(* Logix 5000 project; controller Ex_2_12 Emulate 5570 rev 33.11; software revision 33.00 *)
// Pallet lift table

TASK MainTask (continuous, watchdog 500 ms) : MainProgram

MODULES
   Local : Emulate 5570 (ICP 4, rev 33.11)
END_MODULES

VAR_GLOBAL   (* controller tags *)
   B1 : BOOL;   // Downward Sensor
   B2 : BOOL;   // Upward Sensor
   M1_Downward : BOOL;   // Actuator M1
   M1_Upward : BOOL;   // Actuator M1
   S1 : BOOL;   // Switch S1
   S2 : BOOL;   // Switch S2
END_VAR

PROGRAM MainProgram   (* main routine MainRoutine *)

ROUTINE MainRoutine   (* ladder *)
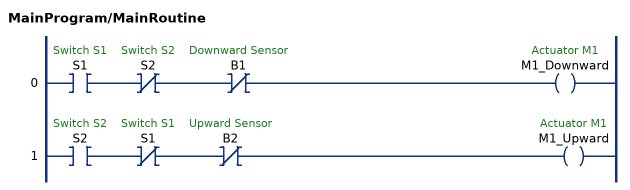
   0: XIC(S1)XIO(S2)XIO(B1)OTE(M1_Downward);
   1: XIC(S2)XIO(S1)XIO(B2)OTE(M1_Upward);
END_ROUTINE
END_PROGRAM
